// TIA Portal project "hm24_iih2iih_simple_production_line" (V19)

(* hardware
DEVICE "S7-1500/ET200MP station_1"  S7-1500 station
   slot 0: "Rail_0"  Rack  6ES7 590-1***0-0AA0
   slot 1: "PLC_1"  CPU 1518-4 PN/DP  6ES7 518-4AP00-0AB0  V3.0
      slot 3: "CPU display_1"  6ES7591-1BA00-0AA0
      slot 32768: "PROFINET interface_1"  X1
         slot 32769: "Port_1"  X1 P1
         slot 32770: "Port_2"  X1 P2
      slot 33024: "PROFINET interface_2"  X2
         slot 33025: "Port_1"  X2 P1
      slot 33280: "PROFINET interface GBIT_3"  X3
         slot 33281: "Port_1"  X3 P1
      slot 33536: "DP interface_1"  X4
      slot 34817: "Virtual CP interface port_1"  Virtual CP interface port  Virtual CP interface port
*)

// ===== PLC "PLC_1"  CPU 1518-4 PN/DP =====

VAR_GLOBAL   // PLC tag table "Default tag table"
   "Packaging_Quality" AT %ID0 : Real;
   "Test_Successful" AT %I4.0 : Bool;
   "Watt_Usage" AT %ID5 : Real;
   "Packages_Consumed" AT %ID10 : Real;
END_VAR

DATA_BLOCK "CircuitBoardAssembly_DB_1"   // DB2
{ S7_Optimized_Access := 'TRUE' }
VERSION : 0.1
// stored: InstanceOfName CircuitBoardAssembly
"CircuitBoardAssembly"
BEGIN
END_DATA_BLOCK

DATA_BLOCK "Enclosure_Assembly_DB_1"   // DB3
{ S7_Optimized_Access := 'TRUE' }
VERSION : 0.1
// stored: InstanceOfName Enclosure_Assembly
"Enclosure_Assembly"
BEGIN
END_DATA_BLOCK

DATA_BLOCK "TestingNPackaging_DB_1"   // DB6
{ S7_Optimized_Access := 'TRUE' }
VERSION : 0.1
// stored: InstanceOfName TestingNPackaging
"TestingNPackaging"
BEGIN
END_DATA_BLOCK

FUNCTION_BLOCK "CircuitBoardAssembly"   // FB1, SCL
{ S7_Optimized_Access := 'TRUE' }
VERSION : 0.1
   VAR
      Soldering_Temperature : Real := 350.0;
      Movement_Speed : Real := 2.0;
      Timestamp : DTL;
      diTime : Real;
      Watt_Usage : Real;
      reset : Bool;
      Circuits_Consumed : Int;
      rRandom : Real;
   END_VAR
   VAR_TEMP
      "temp-retvalRD" : Int;
      "temp-datetime" : Date_And_Time;
   END_VAR
   VAR CONSTANT
      Const_Solder_Temperature : LReal := 350.0;
      Const_kwh_per_sec_Usage : LReal := 0.00278;
      Const_Movement_Speed : LReal := 2.0;
   END_VAR
BEGIN
   // Add randomness to sensor data
   #diTime := USINT_TO_REAL(#Timestamp.SECOND);
   #rRandom := SIN(#diTime) * 0.5;

   #Movement_Speed := #Const_Movement_Speed + #rRandom + 0.7762 ;
   #Soldering_Temperature := #Const_Solder_Temperature + #rRandom  + 0.3802;
   #Watt_Usage := #Const_kwh_per_sec_Usage + #Watt_Usage;
   #Circuits_Consumed := #Circuits_Consumed + 1;

   //Calculate Timestamp
   #"temp-retvalRD" := RD_SYS_T(#"temp-datetime");
   #Timestamp := #"temp-datetime";


   IF #reset = TRUE THEN
       #Watt_Usage := 0;
       #Circuits_Consumed := 0;
       ;
   END_IF;
END_FUNCTION_BLOCK

FUNCTION_BLOCK "Enclosure_Assembly"   // FB2, SCL
{ S7_Optimized_Access := 'TRUE' }
VERSION : 0.1
   VAR
      Enclosure_Pressure : LReal;
      Watt_Usage : LReal;
      Movement_Speed : LReal;
      Timestamp : DTL;
      diTime : Real;
      reset : Bool;
      Enclosures_Consumed : Int;
      rRandom : Real;
   END_VAR
   VAR_TEMP
      "temp-datetime" : Date_And_Time;
      "temp-retvalRD" : Int;
   END_VAR
   VAR CONSTANT
      Const_Enclosure_Pressure : LReal := 20.0;
      Const_kwh_per_sec_Usage : LReal := 0.00378;
      Const_Movement_Speed : LReal := 4.0;
   END_VAR
BEGIN
   // Add randomness to sensor data
   #diTime := USINT_TO_REAL(#Timestamp.SECOND);
   #rRandom := SIN(#diTime) * 0.5;

   #Movement_Speed := #Const_Movement_Speed + #rRandom + 0.5483;
   #Enclosure_Pressure := #Const_Enclosure_Pressure + #rRandom  + 0.6021;
   #Watt_Usage := #Const_kwh_per_sec_Usage + #Watt_Usage;
   #Enclosures_Consumed := #Enclosures_Consumed + 1;

   //Calculate Timestamp
   #"temp-retvalRD" := RD_SYS_T(#"temp-datetime");
   #Timestamp := #"temp-datetime";

   IF #reset = TRUE THEN
       #Watt_Usage := 0;
       #Enclosures_Consumed := 0;
       ;
   END_IF;
END_FUNCTION_BLOCK

FUNCTION_BLOCK "TestingNPackaging"   // FB3, SCL
{ S7_Optimized_Access := 'TRUE' }
VERSION : 0.1
   VAR
      Watt_Usage : Real;
      Packaging_Quality : LReal := 98.0;
      Test_Successful : Bool := True;
      Timestamp : DTL := DTL#1970-01-01-00:00:00;
      diTime : Real;
      Packages_Consumed : Int;
      reset : Bool;
      rRandom : Real;
   END_VAR
   VAR_TEMP
      "temp-datetime" : Date_And_Time;
      "temp-retvalRD" : Int;
   END_VAR
   VAR CONSTANT
      Const_kwh_per_sec_Usage : LReal := 0.00401;
      Const_Packaging_Quality : LReal := 95.0;
   END_VAR
BEGIN
   // Add randomness to sensor data
   #diTime := USINT_TO_REAL(#Timestamp.SECOND);
   #rRandom := SIN(#diTime);

   #Packaging_Quality := #Const_Packaging_Quality + #rRandom  + 0.7372;

   #Watt_Usage := #Const_kwh_per_sec_Usage + #Watt_Usage;



   IF (ABS(#rRandom) > 0.1) THEN
       #Test_Successful := True;
       #Packages_Consumed := #Packages_Consumed + 1;
   ELSE
       #Test_Successful := False;
   END_IF;

   //Calculate Timestamp
   #"temp-retvalRD" := RD_SYS_T(#"temp-datetime");
   #Timestamp := #"temp-datetime";
   "Packaging_Quality" := #Packaging_Quality;
   "Test_Successful" := #Test_Successful;
   "Watt_Usage" := #Watt_Usage;
   "Packages_Consumed" := #Packages_Consumed;

   IF #reset = TRUE THEN
       #Watt_Usage := 0;
       #Packages_Consumed := 0;
       ;
   END_IF;
END_FUNCTION_BLOCK

ORGANIZATION_BLOCK "Main"   // OB1, LAD, ProgramCycle
TITLE = "Main Program Sweep (Cycle)"
{ S7_Optimized_Access := 'TRUE' }
VERSION : 0.1
   VAR_INPUT
      Initial_Call : Bool;   // Initial call of this OB
      Remanence : Bool;   // =True, if remanent data are available
   END_VAR
BEGIN
END_ORGANIZATION_BLOCK

ORGANIZATION_BLOCK "CyclicInterrupt"   // OB30, FBD, CyclicInterrupt
{ S7_Optimized_Access := 'TRUE' }
VERSION : 0.1
   VAR_INPUT
      Initial_Call : Bool;   // Initial call of this OB
      Event_Count : Int;   // Events discarded
   END_VAR
BEGIN

REGION Network 1
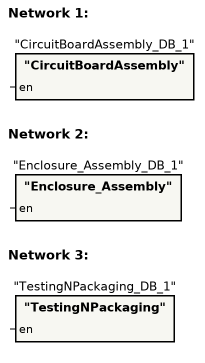
   "CircuitBoardAssembly_DB_1"();   // "CircuitBoardAssembly"
END_REGION

REGION Network 2
   "Enclosure_Assembly_DB_1"();   // "Enclosure_Assembly"
END_REGION

REGION Network 3
   "TestingNPackaging_DB_1"();   // "TestingNPackaging"
END_REGION
END_ORGANIZATION_BLOCK